// TIA Portal V20 export
TYPE "typeSequenceControlNodeJobInterface_transferPnPLeft"
// stored: Namespace Unit1.Em5
   STRUCT
      sideTapePICKJob2_A : "LER_typeJobInterface";
      hotPressLeftPLACEJob3_A : "LER_typeJobInterface";
      hotPressLeftPICKJob4_A : "LER_typeJobInterface";
      sideTapePICKJob5_B : "LER_typeJobInterface";
      hotPressRightPLACEJob6_B : "LER_typeJobInterface";
      hotPressRightPICKJob7_B : "LER_typeJobInterface";
      hipotThicknessPLACEJob9 : "LER_typeJobInterface";
   END_STRUCT;
END_TYPE
